ABB RAPID module: TCP_t2B_final.MOD

MODULE TCP_t2B7
	! Points are read in order of declaration.
  ! Please do not change the order of points!

  LOCAL PERS robtarget pTCP_Point1:=[[517.2705,-5.522776,300.6515],[0.499380886554718,-0.00519778858870268,0.866347849369049,0.00575591530650854],[-1,1,-2,0],[9E+09,9E+09,9E+09,9E+09,9E+09,9E+09]];
	LOCAL PERS robtarget pTCP_Point2:=[[517.4753,26.61037,296.8748],[0.494102329015732,0.329368144273758,0.796000480651855,-0.117314644157887],[0,-2,1,0],[9E+09,9E+09,9E+09,9E+09,9E+09,9E+09]];
	LOCAL PERS robtarget pTCP_Point3:=[[503.4368,-18.01744,289.8195],[0.55969101190567,-0.0462285429239273,0.825725138187408,0.0527913570404053],[-1,-3,2,0],[9E+09,9E+09,9E+09,9E+09,9E+09,9E+09]];
	LOCAL PERS robtarget pTCP_Point4:=[[507.7421,7.820115,294.2143],[0.536838114261627,0.138700500130653,0.83128809928894,-0.0390773229300976],[0,-2,1,0],[9E+09,9E+09,9E+09,9E+09,9E+09,9E+09]];

ENDMODULE
